// TwinCAT 3 PLC project Nepionic_Log_Test
// ProgramVersion: 3.1.4026.20
// libraries:
//   [Nepionic_Log], * (Nepionic)
//   Tc2_Standard, * (Beckhoff Automation GmbH)
//   Tc2_System, * (Beckhoff Automation GmbH)
//   Tc2_TcpIp, * (Beckhoff Automation GmbH)
//   Tc2_Utilities, * (Beckhoff Automation GmbH)
//   Tc3_Module, * (Beckhoff Automation GmbH)
// project tree:
//   Lib/ AnyToString.TcPOU, Constants.TcGVL, DateTime.TcPOU, DeleteFilesState.TcDUT, DeleteOldFiles.TcPOU, DynamicStringBuffer.TcPOU, Error.TcDUT, ErrorCodes.TcDUT, GenerateTimeData.TcPOU, GetFileAgeInSeconds.TcPOU, ILimitedStringBuilder.TcIO, ILog.TcIO, ILogCore.TcIO, IStringBuilder.TcIO, LoggingConfiguration.TcDUT, LogLevel.TcDUT, LogLevelToAdsLogMsgType.TcPOU, PersistToFileState.TcDUT, RollingIntervals.TcDUT, StringBuilder.TcPOU, TcLog.TcPOU, TcLogCore.TcPOU, TcLogTrig.TcPOU
//   Lib/Syslog/ SyslogClient.TcPOU
//   Programs/ TestRunner.TcPOU
//   Tasks/ TestTask.TcTTO
// real-time tasks:
//   TASK PlcTask: cycle T#10ms, priority 20, ADS port 350

CONFIGURATION Nepionic_Log_Test
    RESOURCE PLC ON TwinCAT3
        TASK TestTask(INTERVAL := T#10ms, PRIORITY := 20);
        PROGRAM TestRunner WITH TestTask : TestRunner;
    END_RESOURCE
END_CONFIGURATION

// ---- Lib/DeleteFilesState.TcDUT
// States for state machine used in `DeleteOldFiles`.
{attribute 'qualified_only'}
{attribute 'strict'}
TYPE INTERNAL DeleteFilesState :
(
	Idle := 0,
  SearchNextFile,
  WaitUntilExecutionDone,
  ProcessFoundFiles,
  CheckIfFileIsDirectory,
  CheckFileTime,
  DeleteFile,
  FileDeleted
);
END_TYPE

// ---- Lib/Error.TcDUT
/// This is the error type used in this library.
TYPE Error :
STRUCT
  /// `TRUE` signals an active error
	Active : BOOL;
  /// Error code of type `ErrorCodes`
	Code : INT;
  /// Plain text error message
	Info : Tc2_System.T_MaxString;
END_STRUCT
END_TYPE

// ---- Lib/ErrorCodes.TcDUT
/// Provides error codes for TcLogCore
{attribute 'qualified_only'}
{attribute 'strict'}
{attribute 'to_string'}
TYPE ErrorCodes : 
(
	None := 0,
	OpeningFileFailed,
	WritingToFileFailed,
	ClosingFileFailed,
	EnumeratingFilesInSpecifiedDirectoryFailed,
	DeletingFileFailed,
	FifoOverflow
);
END_TYPE

// ---- Lib/LoggingConfiguration.TcDUT
// Configuration of TcLogCore
TYPE LoggingConfiguration :
STRUCT
	// File name where the logs should be written to. Should not include path.
	file_name : Tc2_System.T_MaxString;
  // File path where the logs should be written to. Will be prefixed to `FileName`
	file_path : Tc2_System.T_MaxString;
  // Whether to include the instance path of TcLog into the log message or not.
	IncludeInstancePath : BOOL;
  /// Whether to write the logs to ADS output or not.
	WriteToAds : BOOL;
  /// Rolling interval: when to create a new log file.
	RollingInterval : RollingIntervals;
  /// What is the minimum log level that gets logged?
	MinimumLevel : LogLevel;
  /// Which delimiter should be used between the different parts of the log string?
	Delimiter : STRING(1);
  /// When should old log files be deleted? Unit: days. Set it to `0` if log files should never be deleted. 
	LogFileLifespan : UINT;
  /// Format of timestamp. See `TcLogCore.TimestampFormat` for formatting options.
	TimestampFormat : STRING;
  /// Log only valid timestamps (skip log messages during time initialization (first few cycles)
  	ValidTimestampsOnly: BOOL;
END_STRUCT
END_TYPE

// ---- Lib/LogLevel.TcDUT
{attribute 'qualified_only'}
{attribute 'strict'}
{attribute 'to_string'}
TYPE LogLevel :
(
	Debug := 0,
	Information,
	Warning,
	Error,
	Fatal
);
END_TYPE

// ---- Lib/PersistToFileState.TcDUT
// States for state machine used in `DynamicStringBuffer.PersistToFile`
{attribute 'qualified_only'}
{attribute 'strict'}
TYPE INTERNAL PersistToFileState :
(
	Idle := 0,
	OpenFile,
	GetStringFromFifo,
	AppendDataToFile,
	CloseFile
);
END_TYPE

// ---- Lib/RollingIntervals.TcDUT
/// Rolling interval to create a new log file when expired. 
{attribute 'qualified_only'}
{attribute 'strict'}
{attrivute 'to_string'}
TYPE RollingIntervals :
(
	None := 0,
	Hourly,
	Daily,
	Monthly
);
END_TYPE

// ---- Lib/Constants.TcGVL
{attribute 'qualified_only'}
VAR_GLOBAL CONSTANT
	/// Fifo overhead needed to manage the string buffer
	FifoOverhead : UDINT := 10;
	/// Buffer size of temporary buffer used to persist all log messages in one cycle. 
	BufferSize : UDINT := (100 * (Tc2_System.MAX_STRING_LENGTH + FifoOverhead));
END_VAR

// ---- Lib/ILimitedStringBuilder.TcIO
{attribute 'hide'}
INTERFACE INTERNAL ILimitedStringBuilder

METHOD Append : IStringBuilder // Append text TO t current build STRING.
VAR_INPUT
    Text : Tc2_System.T_MaxString; //Text to append to current build string
END_VAR
END_METHOD

METHOD AppendIf : IStringBuilder
VAR_INPUT
    Condition : BOOL;
    Text : Tc2_System.T_MaxString;
END_VAR
END_METHOD

METHOD Reset : ILimitedStringBuilder //Reset current build STRING TO an empty STRING.
END_METHOD

METHOD ToString : Tc2_System.T_MaxString //Returns current build STRING.
END_METHOD

END_INTERFACE

// ---- Lib/ILog.TcIO
INTERFACE ILog

METHOD SetLogger : BOOL
VAR_INPUT
    ref2Core : ILogCore;
END_VAR
END_METHOD

END_INTERFACE

// ---- Lib/ILogCore.TcIO
INTERFACE ILogCore EXTENDS __System.IQueryInterface

// Logger method.
// Logs data in custom format. No additional formatting will be done.
METHOD LogCustomFormat : BOOL
VAR_INPUT
    data : Tc2_System.T_MaxString; // Data to be logged. No additional formatting will be done.
END_VAR
END_METHOD

// Logger method.
// Logs in the standard format. This includes
// - timestamp
// - log level
// - log message
// - instance path of logging source (optional)
// The message will only be logged if the logging level exceeds the configured minimum logging level.
METHOD LogStandardFormat : BOOL
VAR_INPUT
    data : Tc2_System.T_MaxString; // Data to be logged. Additional formatting wil be done.
    instancePath : Tc2_System.T_MaxString; // Instance path of calling logger to locate source of logging message.
    logLevel : LogLevels; // Log level of message.
END_VAR
END_METHOD

END_INTERFACE

// ---- Lib/IStringBuilder.TcIO
{attribute 'hide'}
INTERFACE INTERNAL IStringBuilder

METHOD Append : IStringBuilder // Append text TO t current build STRING.
VAR_INPUT
    Text : Tc2_System.T_MaxString; //Text to append to current build string
END_VAR
END_METHOD

METHOD AppendIf : IStringBuilder
VAR_INPUT
    Condition : BOOL;
    Text : Tc2_System.T_MaxString;
END_VAR
END_METHOD

METHOD InsertAtLocation : IStringBuilder
VAR_INPUT
    Text : Tc2_System.T_MaxString;
    Position : INT;
END_VAR
END_METHOD

METHOD PadLeft : IStringBuilder
VAR_INPUT
    text : Tc2_System.T_MaxString; // Text to append to current build string
    length : INT; // Total length of text + padding
    c : STRING(1); // Character to be padded left of text
END_VAR
END_METHOD

METHOD Reset : ILimitedStringBuilder //Reset current build STRING TO an empty STRING.
END_METHOD

METHOD ToString : Tc2_System.T_MaxString //Returns current build STRING.
END_METHOD

END_INTERFACE

// ---- Programs/TestRunner.TcPOU
PROGRAM TestRunner
VAR
	syslogger : SyslogClient(hostname := '127.0.0.1', port := 514);
	
	message : STRING(255) := 'Get a hot dog up ya!';
	send : BOOL;
END_VAR

IF send THEN
	send := FALSE;
	syslogger.SendLog(2, message);
END_IF

syslogger.Execute();

END_PROGRAM

// ---- Lib/Syslog/SyslogClient.TcPOU
FUNCTION_BLOCK SyslogClient
VAR
	// Properties
	_hostname : STRING := '127.0.0.1';
	_port : UINT := 514;
	app_name : STRING(32) := 'TwinCAT_PLC';
    
	// Internal Logic
	socket_handle : Tc2_TcpIp.T_HSocket;
	socket_create : Tc2_TcpIp.Fb_SocketUdpCreate;
	udp_send : Tc2_TcpIp.Fb_SocketUdpSendTo;
    
    log_payload : STRING(512);
    timestamp : STRING(32);
    get_time : Tc2_Utilities.NT_GetTime;
    
    state : INT := 0;
END_VAR

PROPERTY PUBLIC AppName : STRING(255)
GET // PUBLIC
AppName := app_name;
END_GET
SET // PUBLIC
app_name := AppName;
END_SET
END_PROPERTY

METHOD PUBLIC Execute
CASE state OF
    0: // Idle
        
    10: // Fetch Timestamp
        get_time(START := TRUE);
        IF NOT get_time.BUSY AND NOT get_time.ERR THEN
            UpdateTimestamp();
            get_time(START := FALSE);
            state := 20;
        ELSIF get_time.ERR THEN
            get_time(START := FALSE);
            state := 0;
        END_IF

    20: // Maintain Socket
        IF socket_handle.handle = 0 THEN
			socket_create(
				bExecute := TRUE,
				sLocalHost := _hostname,
				nLocalPort := 4444
			);
			IF NOT socket_create.bBusy AND NOT socket_create.bError THEN
				socket_handle := socket_create.hSocket;
				socket_create(bExecute := FALSE);
			END_IF
		ELSE
			state := 30;
		END_IF

    30: // Dispatch UDP
        udp_send(
            hSocket := socket_handle, 
            sRemoteHost := _hostname, 
            nRemotePort := _port,
            pSrc := ADR(log_payload), 
            cbLen := INT_TO_UDINT(Tc2_Standard.Len(log_payload)), 
            bExecute := TRUE
		);
            
        IF NOT udp_send.bBusy AND NOT udp_send.bError THEN
            udp_send(bExecute := FALSE);
            state := 0; 
        END_IF
END_CASE
END_METHOD

//FB_Init is always available implicitly and it is used primarily for initialization.
//The return value is not evaluated. For a specific influence, you can also declare the
//methods explicitly and provide additional code there with the standard initialization
//code. You can evaluate the return value.
METHOD FB_Init: BOOL
VAR_INPUT
    bInitRetains: BOOL; // TRUE: the retain variables are initialized (reset warm / reset cold)
    bInCopyCode: BOOL;  // TRUE: the instance will be copied to the copy code afterward (online change)
	hostname : STRING(15);
	port : UINT;   
END_VAR
THIS^._hostname := hostname;
THIS^._port := port;
END_METHOD

PROPERTY PUBLIC Hostname : STRING(15)
GET // PUBLIC
Hostname := _hostname;
END_GET
SET // PUBLIC
_hostname := Hostname;
ResetConnection();
END_SET
END_PROPERTY

PROPERTY PUBLIC Port : UINT
GET // PUBLIC
Port := _port;
END_GET
SET // PUBLIC
_port := Port;
ResetConnection();
END_SET
END_PROPERTY

METHOD PRIVATE ResetConnection
END_METHOD

METHOD PUBLIC SendLog
VAR_INPUT
    severity : INT; // 0: Emerg ... 7: Debug
    message  : STRING(255);
END_VAR
VAR_INST
    priority : INT;
END_VAR
// Facility 1 (User) * 8 + severity
priority := 8 + severity;

// Build RFC 5424 String: <PRI>1 TIMESTAMP HOSTNAME APPNAME - - - MESSAGE
log_payload := Tc2_System.Concat('<', INT_TO_STRING(priority));
log_payload := Tc2_System.Concat(log_payload, '>1 ');
log_payload := Tc2_System.Concat(log_payload, timestamp);
log_payload := Tc2_System.Concat(log_payload, ' ');
log_payload := Tc2_System.Concat(log_payload, hostname);
log_payload := Tc2_System.Concat(log_payload, ' ');
log_payload := Tc2_System.Concat(log_payload, app_name);
log_payload := Tc2_System.Concat(log_payload, ' - - - ');
log_payload := Tc2_System.Concat(log_payload, message);

state := 10;
END_METHOD

METHOD PRIVATE UpdateTimestamp
timestamp := WORD_TO_STRING(get_time.TimeStr.wYear);
timestamp := Tc2_System.Concat(timestamp, '-');
timestamp := Tc2_System.Concat(timestamp, Tc2_System.RIGHT(Tc2_System.Concat('0', WORD_TO_STRING(get_time.TimeStr.wMonth)), 2));
timestamp := Tc2_System.Concat(timestamp, '-');
timestamp := Tc2_System.Concat(timestamp, Tc2_System.RIGHT(Tc2_System.Concat('0', WORD_TO_STRING(get_time.TimeStr.wDay)), 2));
timestamp := Tc2_System.Concat(timestamp, 'T');
timestamp := Tc2_System.Concat(timestamp, Tc2_System.RIGHT(Tc2_System.Concat('0', WORD_TO_STRING(get_time.TimeStr.wHour)), 2));
timestamp := Tc2_System.Concat(timestamp, ':');
timestamp := Tc2_System.Concat(timestamp, Tc2_System.RIGHT(Tc2_System.Concat('0', WORD_TO_STRING(get_time.TimeStr.wMinute)), 2));
timestamp := Tc2_System.Concat(timestamp, ':');
timestamp := Tc2_System.Concat(timestamp, Tc2_System.RIGHT(Tc2_System.Concat('0', WORD_TO_STRING(get_time.TimeStr.wSecond)), 2));
timestamp := Tc2_System.Concat(timestamp, 'Z');
END_METHOD

END_FUNCTION_BLOCK

// ---- Lib/AnyToString.TcPOU
/// Converts value of input data to string, where the input type can be any of 
/// the standard data types.
FUNCTION PUBLIC AnyToString : Tc2_System.T_MaxString
VAR_INPUT
	data : ANY;
END_VAR
VAR
	_any_byte : POINTER TO BYTE;
	_any_usint : POINTER TO USINT;
	_any_int : POINTER TO INT;
	_any_uint : POINTER TO UINT;
	_any_udInt : POINTER TO UDINT;
	_any_sint : POINTER TO SINT;
	_any_dint : POINTER TO DINT;
	_any_lint : POINTER TO LINT;
	_any_ulint : POINTER TO ULINT;
	_any_word : POINTER TO WORD;
	_any_lword : POINTER TO LWORD;
	_any_real : POINTER TO REAL;
	_any_lreal : POINTER TO LREAL;
	_any_date_and_time : POINTER TO DATE_AND_TIME;
	_any_date : POINTER TO DATE;
	_any_time : POINTER TO TIME;
	_any_wstring : POINTER TO WSTRING;
	_any_time_of_day : POINTER TO TOD;
	_any_string : POINTER TO STRING;
	_string : Tc2_System.T_MaxString;
	_wstring : WSTRING;
END_VAR

IF data.TypeClass = __SYSTEM.Type_Class.Type_Byte THEN
	_any_byte := data.pValue;
	AnyToString := BYTE_TO_STRING(_any_byte^);
ELSIF data.TypeClass = __SYSTEM.Type_Class.Type_Int THEN
	_any_int := data.pValue;
	AnyToString := INT_TO_STRING(_any_int^);
ELSIF data.TypeClass = __SYSTEM.Type_Class.Type_UInt THEN
	_any_uint := data.pValue;
	AnyToString := UINT_TO_STRING(_any_uint^);
ELSIF data.TypeClass = __SYSTEM.Type_Class.Type_UDint THEN
	_any_udint := data.pValue;
	AnyToString := UDINT_TO_STRING(_any_udint^);
ELSIF data.TypeClass = __SYSTEM.Type_Class.Type_SInt THEN
	_any_sint := data.pValue;
	AnyToString := SINT_TO_STRING(_any_sint^);
ELSIF data.TypeClass = __SYSTEM.Type_Class.Type_USint THEN
	_any_usint := data.pValue;
	AnyToString := USINT_TO_STRING(_any_usint^);
ELSIF data.TypeClass = __SYSTEM.Type_Class.Type_DInt THEN
	_any_dint := data.pValue;
	AnyToString := DINT_TO_STRING(_any_dint^);
ELSIF data.TypeClass = __SYSTEM.Type_Class.Type_LInt THEN
	_any_lint := data.pValue;
	AnyToString := LINT_TO_STRING(_any_lint^);
ELSIF data.TypeClass = __SYSTEM.Type_Class.Type_ULint THEN
	_any_ulint := data.pValue;
	AnyToString := ULINT_TO_STRING(_any_ulint^);
ELSIF data.TypeClass = __SYSTEM.Type_Class.Type_Word THEN
	_any_word := data.pValue;
	AnyToString := WORD_TO_STRING(_any_word^);
ELSIF data.TypeClass = __SYSTEM.Type_Class.Type_LWord THEN
	_any_lword := data.pValue;
	AnyToString := LWORD_TO_STRING(_any_lword^);
ELSIF data.TypeClass = __SYSTEM.Type_Class.Type_Real THEN
	_any_real := data.pValue;
	AnyToString := REAL_TO_STRING(_any_real^);
ELSIF data.TypeClass = __SYSTEM.Type_Class.Type_LReal THEN
	_any_lreal := data.pValue;
	AnyToString := LREAL_TO_STRING(_any_lreal^);
ELSIF data.TypeClass = __SYSTEM.Type_Class.Type_DateAndTime THEN
	_any_date_and_time := data.pValue;
	AnyToString := DT_TO_STRING(_any_date_and_time^);  
ELSIF data.TypeClass = __SYSTEM.Type_Class.Type_Date THEN
	_any_date := data.pValue;
	AnyToString := DATE_TO_STRING(_any_date^);
ELSIF data.TypeClass = __SYSTEM.Type_Class.Type_Time THEN
	_any_time := data.pValue;
	AnyToString := TIME_TO_STRING(_any_time^);
ELSIF data.TypeClass = __SYSTEM.Type_Class.Type_String THEN
	_any_string := data.pValue;
	AnyToString := _any_string^;
ELSIF data.TypeClass = __SYSTEM.Type_Class.Type_WString THEN
	_any_wstring := data.pValue;
	_wString := _any_wstring^;
	Tc2_Utilities.WSTRING_TO_STRING2(ADR(_string), ADR(_wstring), SIZEOF(_wstring));
	AnyToString := _string;
ELSIF data.TypeClass = __SYSTEM.Type_Class.Type_TimeOfDay THEN
	_any_time_of_day := data.pValue;
	AnyToString := TOD_TO_STRING(_any_time_of_day^);
ELSE
	AnyToString := TO_STRING(data.pValue^);
END_IF

END_FUNCTION

// ---- Lib/DateTime.TcPOU
/// Generate time data in different formats.
{attribute: 'hide_all_locals'}
FUNCTION_BLOCK PUBLIC DateTime
VAR
  local_system_time : Tc2_Utilities.FB_LocalSystemTime;
  get_system_time : Tc2_System.GetSystemTime;
  time_zone_info : Tc2_Utilities.FB_GetTimeZoneInformation;
  local_Time : Tc2_Utilities.FB_SystemTimeToTzSpecificLocalTime;
  local_system_time_valid : Tc2_Standard.R_Trig;
  utc_time : Tc2_Utilities.FB_TzSpecificLocalTimeToFileTime;
END_VAR

// Get local system time
local_system_time(
	sNetID  :=  '',
	bEnable :=  TRUE,
	dwCycle :=  1,
	dwOpt :=  1,
	tTimeout:= Tc2_System.Default_Ads_Timeout
);

// Get timezone information
time_zone_info(
	sNetID := '',
	bExecute := TRUE,
	tTimeout := Tc2_System.Default_Ads_Timeout
);

// Convert local time to utc time
utc_time(
	in := THIS^.AsLocalFileTime,
	tzInfo := time_zone_info.tzInfo
);
  
// Finished retrieving time data
local_system_time_valid(Clk := local_system_time.bValid);

/// Returns local time as `Tc2_Utilities.T_FILETIME`.
{attribute 'monitoring':='variable'}
PROPERTY AsLocalFileTime : Tc2_Utilities.T_FILETIME
GET
AsLocalFileTime := SYSTEMTIME_TO_FILETIME(THIS^.AsLocalSystemTime);
END_GET
END_PROPERTY

/// Returns local time as `Tc2_Utilities.TIMESTRUCT`.
{attribute 'monitoring':='variable'}
PROPERTY AsLocalSystemTime : Tc2_Utilities.TIMESTRUCT
GET
AsLocalSystemTime := local_system_time.systemTime;
END_GET
END_PROPERTY

/// Returns local time as string.
{attribute 'monitoring':='variable'}
PROPERTY AsLocalSystemTimeString : Tc2_System.T_MAXSTRING
GET
AsLocalSystemTimeString := Tc2_Utilities.SYSTEMTIME_TO_STRING(THIS^.AsLocalSystemTime);
END_GET
END_PROPERTY

/// Returns UTC time as `Tc2_Utilities.T_FILETIME`.
{attribute 'monitoring':='variable'}
PROPERTY AsUtcFileTime : Tc2_Utilities.T_FILETIME
GET
AsUtcFileTime := utc_time.out;
END_GET
END_PROPERTY

/// When calling `DateTime` the first time, it takes some time until all time and timezone information is available.
/// `Done` is `TRUE` for one cycle, once all the data is ready. 
{attribute 'monitoring':='call'}
PROPERTY Done : BOOL
GET
Done := local_system_time_valid.Q;
END_GET
END_PROPERTY

// Replaces placeholders in format string by the actual time values.
{attribute 'hide_all_locals'}
{attribute 'hide'}
METHOD PRIVATE ReplaceFormatPlaceholder : STRING
VAR_INPUT
  format : STRING;
  length : INT;
  timeType : STRING(1);
END_VAR
VAR_INST
  i : INT;
  replaceString : STRING;
  timeString : STRING;
END_VAR
VAR
  localSystemTime : Tc2_Utilities.TIMESTRUCT;
END_VAR
localSystemTime := THIS^.AsLocalSystemTime;

IF    timeType = 'Y'  THEN timeString := TO_STRING(localSystemTime.wYear); 
ELSIF timeType = 'M'  THEN timeString := TO_STRING(localSystemTime.wMonth); 
ELSIF timeType = 'D'  THEN timeString := TO_STRING(localSystemTime.wDay); 
ELSIF timeType = 'h'  THEN timeString := TO_STRING(localSystemTime.wHour); 
ELSIF timeType = 'm'  THEN timeString := TO_STRING(localSystemTime.wMinute); 
ELSIF timeType = 's'  THEN timeString := TO_STRING(localSystemTime.wSecond); 
ELSIF timeType = 'i'  THEN timeString := TO_STRING(localSystemTime.wMilliseconds); 
ELSE
  timeString:='';
END_IF

replaceString := '';

IF length > Tc2_Standard.LEN(timeString) THEN
  FOR i:=1 TO length - Tc2_Standard.LEN(timeString) DO
    replaceString := Tc2_Standard.CONCAT(replaceString, '0');
  END_FOR
  replaceString := Tc2_Standard.CONCAT(replaceString, timeString);
ELSE
  replaceString := Tc2_Standard.RIGHT(timeString, length);
END_IF

ReplaceFormatPlaceholder := Tc2_Standard.REPLACE(format, replaceString, length, Tc2_Standard.FIND(format, timeType));
END_METHOD

/// Returns a formatted string containing the actual time information 
/// - `Y` : year
/// - `M` : month
/// - `D` : day
/// - `h` : hour 
/// - `m` : minute
/// - `s` : second
/// - `i` : millisecond
/// 
/// Example:    
/// _YYMMDD-hh:mm:ss:iii_   
/// => _20210812-12:30:22:123_
{attribute 'hide_all_locals'}
METHOD ToFormatString : Tc2_System.T_MaxString
VAR_INPUT
  /// Format the timestamp should have.
  format : STRING;
END_VAR
VAR_INST
  inputString : STRING;
  c : STRING(1);
  formattedString : Tc2_System.T_MaxString;
END_VAR
VAR
  year : INT := 0;
  month : INT := 0;
  day : INT := 0;
  hour : INT := 0;
  minute : INT := 0;
  second : INT := 0;
  millisecond : INT := 0;
END_VAR
VAR CONSTANT
  ValidFormat : STRING := 'YMDhms';
END_VAR
// Parses "format" and returns a adequatly formatted string containing the time information
inputString := format;

WHILE Tc2_Standard.LEN(inputString) > 0 DO
  c := Tc2_Standard.LEFT(inputString, 1);
  
  IF    c = 'Y' THEN year := year + 1;
  ELSIF c = 'M' THEN month := month + 1;
  ELSIF c = 'D' THEN day := day + 1;
  ELSIF c = 'h' THEN hour := hour + 1;
  ELSIF c = 'm' THEN minute := minute + 1;
  ELSIF c = 's' THEN second := second + 1;
  ELSIF c = 'i' THEN millisecond := millisecond + 1;
  END_IF
  
  inputString := Tc2_Standard.DELETE(inputString, 1, 1);
END_WHILE

formattedString := ReplaceFormatPlaceholder(format, year, 'Y');
formattedString := ReplaceFormatPlaceholder(formattedString, month, 'M');
formattedString := ReplaceFormatPlaceholder(formattedString, day, 'D');
formattedString := ReplaceFormatPlaceholder(formattedString, hour, 'h');
formattedString := ReplaceFormatPlaceholder(formattedString, minute, 'm');
formattedString := ReplaceFormatPlaceholder(formattedString, second, 's');
formattedString := ReplaceFormatPlaceholder(formattedString, millisecond, 'i');

ToFormatString := formattedString;
END_METHOD

END_FUNCTION_BLOCK

// ---- Lib/DeleteOldFiles.TcPOU
{attribute 'hide_all_locals'}
FUNCTION_BLOCK INTERNAL DeleteOldFiles
VAR_INPUT
  StartScan : BOOL; // Rising edge starts scan for out-of-date log files and deletes them.
  ExpirationInDays : UINT; // Files will be deleted if older than n days
  FilePath : Tc2_System.T_MaxString; // Path to files to be deleted
  FileName : Tc2_System.T_MaxString; // Only files which match this filename will be deleted
  CurrentUtcTime : Tc2_Utilities.T_FILETIME; // Current time  as UTC
END_VAR
VAR_OUTPUT
  Error : Error; // Error information
END_VAR
VAR CONSTANT
  OneDayInSeconds : LREAL := 24*3600.0;
  MaxNumberOfFiles : UDINT := 100;
END_VAR
VAR
  _state : DeleteFilesState := DeleteFilesState.Idle;
  
  _enumFindFileList : Tc2_Utilities.FB_EnumFindFileList;
  _enumBusy : Tc2_Standard.F_TRIG;
  _fileDelete : Tc2_System.FB_FileDelete;
  _fileDeleteBusy : Tc2_Standard.F_TRIG;
  _listOfFiles : ARRAY[1..100] OF Tc2_Utilities.ST_FindFileEntry;
  _deleteFileIndex : UDINT;
  _fileNameToDelete : Tc2_System.T_MaxString;
  _commandType : Tc2_Utilities.E_EnumCmdType;
  _fileDeleted : BOOL;
  _startFileDelete: BOOL;
END_VAR

// State machine to delete all due files.
// It first enumerates all files in the specified directory
// and then deletes all files that have overpassed the specified due date
_startFileDelete := FALSE;

CASE _state OF
  DeleteFilesState.Idle:
    IF StartScan THEN
      _commandType:= eEnumCmd_First;
      _deleteFileIndex := 1;
      _state := DeleteFilesState.SearchNextFile;
    END_IF
    
  DeleteFilesState.SearchNextFile:
    IF _enumBusy.Q THEN
      _state := DeleteFilesState.WaitUntilExecutionDone;
    END_IF
    
  DeleteFilesState.WaitUntilExecutionDone:
    IF NOT _enumFindFileList.bError THEN
      IF NOT _enumFindFileList.bEOE THEN
        IF _enumFindFileList.nFindFiles < MaxNumberOfFiles THEN
          _state := DeleteFilesState.SearchNextFile;
        ELSE
          _commandType := eEnumCmd_Abort;
          _state := DeleteFilesState.ProcessFoundFiles;
        END_IF
      ELSE
        _state := DeleteFilesState.ProcessFoundFiles;
      END_IF
    ELSE
      _state := DeleteFilesState.Idle;
    END_IF
    
  DeleteFilesState.ProcessFoundFiles:
    IF _deleteFileIndex > _enumFindFileList.nFindFiles THEN
      _state := DeleteFilesState.Idle;
    ELSE
      _state := DeleteFilesState.CheckIfFileIsDirectory;
    END_IF
    
  DeleteFilesState.CheckIfFileIsDirectory:
    IF NOT _listOfFiles[_deleteFileIndex].fileAttributes.bDirectory THEN
      _state := DeleteFilesState.CheckFileTime;
    ELSE
      _deleteFileIndex := _deleteFileIndex + 1;
      _state := DeleteFilesState.ProcessFoundFiles;
    END_IF
    
  DeleteFilesState.CheckFileTime:   
    IF GetFileAgeInSeconds(CurrentUtcTime, _listOfFiles[_deleteFileIndex]) > (ExpirationInDays * OneDayInSeconds) THEN
      _state := DeleteFilesState.DeleteFile;
    ELSE
      _deleteFileIndex := _deleteFileIndex + 1;
      _state := DeleteFilesState.ProcessFoundFiles;
    END_IF
  
  DeleteFilesState.DeleteFile:
    _fileNameToDelete := Tc2_Standard.CONCAT(FilePath, _listOfFiles[_deleteFileIndex].sFileName);
    _startFileDelete := TRUE;
    
    IF _fileDeleteBusy.Q THEN
      _deleteFileIndex := _deleteFileIndex + 1;
      _fileDeleted := TRUE;
      _state := DeleteFilesState.FileDeleted;
    END_IF
    IF _fileDelete.bError THEN
      _state := DeleteFilesState.Idle;
    END_IF
    
  DeleteFilesState.FileDeleted:   
    // This state is needed to generate a rising edge for FB_FileDelete
    IF NOT _fileDeleted THEN
      _state := DeleteFilesState.ProcessFoundFiles;
    END_IF
    _fileDeleted := FALSE;

END_CASE

// Function blocks used in state machine

// Search files in given directory
_enumFindFileList(sNetId := '',
       eCmd := _commandType,
       sPathName := Tc2_Standard.CONCAT(FilePath, Tc2_Standard.CONCAT('*', FileName)),
       bExecute := (_state = DeleteFilesState.SearchNextFile) OR (_commandType = eEnumCmd_Abort AND _state <> DeleteFilesState.Idle),
       pFindList := ADR(_listOfFiles),
       cbFindList := SIZEOF(_listOfFiles),
       tTimeout := T#10S);
       
_enumBusy(CLK:=_enumFindFileList.bBusy);

// Delete files
_fileDelete(sNetId := '',
             sPathName := _fileNameToDelete,
             bExecute := _startFileDelete,
             tTimeout := T#10S);

_fileDeleteBusy(CLK := _fileDelete.bBusy);

// Error handling
Error.Active := FALSE;
Error.Code := ErrorCodes.None;
Error.Info := '';

IF _enumFindFileList.bError THEN
  Error.Active := TRUE;
  Error.Code := ErrorCodes.EnumeratingFilesInSpecifiedDirectoryFailed;
  Error.Info := Tc2_Standard.CONCAT('Enumerating files in specified directory failed. Error thrown by FB_EnumFindFileList. Consult Beckhoff InfoSys. Internal Error: ', UDINT_TO_STRING(_enumFindFileList.nErrId));
END_IF
      
IF _fileDelete.bError THEN
  Error.Active := TRUE;
  Error.Code := ErrorCodes.DeletingFileFailed;
  Error.Info := Tc2_Standard.CONCAT('Deleting expired log file in specified directory failed. Error thrown by FB_FileDelete. Consult Beckhoff InfoSys. Internal Error: ', UDINT_TO_STRING(_fileDelete.nErrId));
END_IF

END_FUNCTION_BLOCK

// ---- Lib/GetFileAgeInSeconds.TcPOU
{attribute 'hide'}
FUNCTION INTERNAL GetFileAgeInSeconds : DINT
VAR_INPUT
  currentUtcTime : Tc2_Utilities.T_FILETIME;
  findFileEntry : Tc2_Utilities.ST_FindFileEntry;
END_VAR
VAR
  _timeLastWriteAccess : Tc2_Utilities.T_ULARGE_INTEGER;
  _fileTimeAsULINT : Tc2_Utilities.T_ULARGE_INTEGER;
  _fileTimeDifference : Tc2_Utilities.T_ULARGE_INTEGER;
END_VAR
VAR CONSTANT
  OneSecondInOneHundredNanoSecondsIntervals : LREAL := 1000*1000*10;
END_VAR

// Local file time
_fileTimeAsULINT.dwLowPart := currentUtcTime.dwLowDateTime;
_fileTimeAsULINT.dwHighPart := currentUtcTime.dwHighDateTime;

// Write access is UTC
_timeLastWriteAccess.dwLowPart := findFileEntry.lastWriteTime.dwLowDateTime;
_timeLastWriteAccess.dwHighPart := findFileEntry.lastWriteTime.dwHighDateTime;
_fileTimeDifference := UInt64Sub64(_fileTimeAsULINT, _timeLastWriteAccess);

GetFileAgeInSeconds := LREAL_TO_DINT(UINT64_TO_LREAL(_fileTimeDifference)/(OneSecondInOneHundredNanoSecondsIntervals));

END_FUNCTION

// ---- Lib/DynamicStringBuffer.TcPOU
{attribute 'hide_all_locals'}
FUNCTION_BLOCK INTERNAL DynamicStringBuffer
VAR_OUTPUT
  Error : Error; // Error information of this FB
END_VAR
VAR
  _fifo : Tc2_Utilities.FB_StringRingBuffer; // Necessary to buffer log data until it has been written to file.
  _memoryManager : Tc3_DynamicMemory.FB_DynMem_Manager; // Memory manager, required by DynMem_Buffer.
  _dynamicMemoryBuffer : Tc3_DynamicMemory.FB_DynMem_Buffer(ipMemMan := _memoryManager); // Provides dynamic buffer for Fifo. Is extended automatically if more than the
                                                                   // default buffer size is needed.                  
  _busy : BOOL; // Buffer is busy; typically with writing data to the file system.
END_VAR

METHOD AddLine : BOOL
VAR_INPUT
  text : Tc2_System.T_MaxString; // Text to be added to the buffer
END_VAR
ResizeFifoBufferIfNecessary();
_fifo.A_AddTail(putValue := Tc2_Standard.CONCAT(Tc2_Standard.LEFT(text, 254), '$N'));
END_METHOD

METHOD AddString : BOOL
VAR_INPUT
  text : Tc2_System.T_MaxString; // String to be added to the buffer
END_VAR
ResizeFifoBufferIfNecessary();
_fifo.A_AddTail(putValue := text);
END_METHOD

METHOD PRIVATE AllocateBuffer : BOOL // Allocates buffer FOR the fifo.
VAR_INPUT
  bufferSize : UDINT; // Initial buffer size in BYTEs for fifo buffer.
END_VAR
_dynamicMemoryBuffer.CreateBuffer(nSize:=bufferSize, bReset:=TRUE);
_fifo.pBuffer := _dynamicMemoryBuffer.pBuffer;
_fifo.cbBuffer := bufferSize;
END_METHOD

{attribute 'monitoring':='call'}
PROPERTY Busy : BOOL
GET
Busy := _busy;
END_GET
SET // PRIVATE
_busy := Busy;
END_SET
END_PROPERTY

METHOD FB_exit : BOOL
VAR_INPUT
  bInCopyCode : BOOL; // if TRUE, the exit method is called for exiting an instance that is copied afterwards (online change).
END_VAR
_dynamicMemoryBuffer.Clear();
END_METHOD

METHOD FlushCache : BOOL
_fifo.A_Reset();
END_METHOD

METHOD INTERNAL Init : BOOL
VAR_INPUT
  bufferSize : UDINT; // Initial buffer size in BYTEs for fifo buffer.
END_VAR
AllocateBuffer(bufferSize);
END_METHOD

{attribute 'hide_all_locals'}
METHOD PersistToFile : BOOL
VAR_INPUT
  enable: BOOL; // TRUE starts persistence mechanism
  fileName : Tc2_System.T_MaxString; // File name including its path
END_VAR
VAR_INST
  state : PersistToFileState;
  
  fileOpen : Tc2_System.FB_FileOpen;
  fileHandle : UINT;
  
  fileWrite : Tc2_System.FB_FileWrite;
  lockFileWriteToForceRisingEdge : BOOL; // filePuts can only be executed every other cycle
                                         // since it needs a rising edge to execute.
  fileClose : Tc2_System.FB_FileClose;
  
  buffer : ARRAY[0..CONSTANTS.BufferSize] OF BYTE;
  currentBufferPos : UDINT;
  fifoHeadString : Tc2_System.T_MaxString;
  fifoHeadLength : UDINT;
  fifoHeadBytes : ARRAY[0..Tc2_System.MAX_STRING_LENGTH] OF BYTE;
  i : UINT;
END_VAR
VAR CONSTANT
  NetId : STRING := '';
  Timeout : TIME := DEFAULT_ADS_TIMEOUT;
  MaxLogsPerCycle : UINT := UDINT_TO_UINT(CONSTANTS.BufferSize / Tc2_System.MAX_STRING_LENGTH);
  MaxBufferPosition : UDINT := (SIZEOF(buffer)-Tc2_System.MAX_STRING_LENGTH);
END_VAR
// State machine
// Using if-statements instead of case for performance reasons:
// Some states execute instantly and allow thus the next state 
// to start within the same plc cycle.

// *** I D L E ***
IF state = PersistToFileState.Idle THEN
  lockFileWriteToForceRisingEdge := FALSE;
  IF _fifo.nCount > 0 AND enable THEN 
    lockFileWriteToForceRisingEdge := FALSE;
    state := PersistToFileState.OpenFile;
  END_IF
END_IF
    
// *** O P E N   F I L E ***
fileOpen(sNetId := NetId, sPathName := fileName, nMode := FOPEN_MODEAPPEND OR FOPEN_MODETEXT, 
           ePath := PATH_GENERIC, bExecute := (state = PersistToFileState.OpenFile), tTimeout := Timeout,
           hFile => fileHandle);

IF state = PersistToFileState.OpenFile THEN
  IF fileOpen.bError THEN
    state := PersistToFileState.CloseFile;
  ELSIF NOT fileOpen.bBusy THEN
    state := PersistToFileState.GetStringFromFifo; 
  END_IF
END_IF 

// *** P O P   F R O M   F I F O ***
IF state = PersistToFileState.GetStringFromFifo THEN
  IF NOT lockFileWriteToForceRisingEdge THEN
    currentBufferPos := 0;
    FOR i:=0 TO MaxLogsPerCycle DO
      IF _fifo.nCount <= 0 THEN EXIT; END_IF
      IF currentBufferPos >= MaxBufferPosition THEN EXIT; END_IF
      
      _fifo.A_RemoveHead(getValue => fifoHeadString); 
      fifoHeadBytes := MAXSTRING_TO_BYTEARR(fifoHeadString);
      fifoHeadLength := INT_TO_UDINT(LEN(fifoHeadString));
      MEMCPY(
        destAddr  :=  ADR(buffer) + SIZEOF(BYTE) * currentBufferPos,
        srcAddr   :=  ADR(fifoHeadBytes),
        n     :=  fifoHeadLength);    
      currentBufferPos := currentBufferPos + fifoHeadLength;  
    END_FOR
    state := PersistToFileState.AppendDataToFile;
  END_IF
  lockFileWriteToForceRisingEdge := FALSE;
END_IF
  
// *** W R I T E   T O   F I L E ***
fileWrite(
  sNetId := NetId, 
  hFile := fileHandle, 
  pWriteBuff := ADR(buffer),
  cbWriteLen := currentBufferPos,
  bExecute := state = PersistToFileState.AppendDataToFile, 
  tTimeout := Timeout); 

IF state = PersistToFileState.AppendDataToFile THEN
  lockFileWriteToForceRisingEdge := TRUE;   
  IF fileWrite.bError THEN
    state := PersistToFileState.CloseFile;
  ELSIF _fifo.nCount > 0 AND NOT fileWrite.bBusy THEN
    state := PersistToFileState.GetStringFromFifo; 
  ELSIF _fifo.nCount = 0 THEN
    state := PersistToFileState.CloseFile;
  END_IF
END_IF
    
// *** C L O S E   F I L E ***
fileClose(
  sNetId := NetId, hFile := fileHandle, 
  bExecute := (state = PersistToFileState.CloseFile), tTimeout := Timeout);

IF state = PersistToFileState.CloseFile THEN
  IF NOT fileClose.bBusy THEN state := PersistToFileState.Idle; END_IF
END_IF

// Close file in case of error
IF fileOpen.bError THEN state := PersistToFileState.CloseFile; END_IF
IF fileWrite.bError THEN state := PersistToFileState.CloseFile; END_IF
IF NOT _fifo.bOk AND _fifo.nCount > 0 AND state <> PersistToFileState.Idle THEN 
  state := PersistToFileState.CloseFile; 
END_IF

// Error handling
IF fileOpen.bError THEN
  Error.Active := TRUE;
  Error.Code := ErrorCodes.OpeningFileFailed;
  Error.Info := Tc2_Standard.CONCAT('Opening file failed. Error thrown by FB_FileOpen. Consult Beckhoff InfoSys. Internal Error: ', UDINT_TO_STRING(fileOpen.nErrId));
ELSIF fileWrite.bError THEN
  Error.Active := TRUE;
  Error.Code := ErrorCodes.WritingToFileFailed;
  Error.Info := Tc2_Standard.CONCAT('Writing to file failed. Error thrown by FB_FileWrite. Consult Beckhoff InfoSys. Internal Error: ', UDINT_TO_STRING(fileWrite.nErrId));
ELSIF fileClose.bError THEN
  Error.Active := TRUE;
  Error.Code := ErrorCodes.ClosingFileFailed;
  Error.Info := Tc2_Standard.CONCAT('Closing file failed. Error thrown by FB_FileClose. Consult Beckhoff InfoSys. Internal Error: ', UDINT_TO_STRING(fileClose.nErrId));
ELSIF NOT _fifo.bOk AND _fifo.nCount > 0 THEN
  Error.Active := TRUE;
  Error.Code := ErrorCodes.FifoOverflow;
  Error.Info := 'FIFO overflow. Check if plc has enough free memory.';
ELSE
  Error.Active := FALSE;
  Error.Code := ErrorCodes.None;
  Error.Info := '';
END_IF

// Set busy state
Busy := (state <> PersistToFileState.Idle OR _fifo.nCount > 0);

(* Uncomment for cyclic logging of state machine, buffer usage & errors

ADSLOGSTR(ADSLOG_MSGTYPE_LOG, 
  Tc2_Standard.CONCAT('****DynamicStringBuffer.state:', 
  Tc2_Standard.CONCAT(UINT_TO_STRING(state),
  Tc2_Standard.CONCAT(', DynamicStringBuffer.hFile:', UINT_TO_STRING(hFile)))), '');

ADSLOGSTR(ADSLOG_MSGTYPE_LOG, 
  Tc2_Standard.CONCAT('****Fifo: used ', 
  Tc2_Standard.CONCAT(UDINT_TO_STRING(Fifo.cbSize),
  Tc2_Standard.CONCAT(' of ', UDINT_TO_STRING(Fifo.cbBuffer)))), '');
  
IF Error.Active THEN
  ADSLOGSTR(ADSLOG_MSGTYPE_LOG, 
    Tc2_Standard.CONCAT('****DynamicStringBuffer.Error: ', Error.Info), 
    '');  
END_IF
*)
END_METHOD

METHOD PopHead : Tc2_System.T_MaxString
VAR_INST
  headString : Tc2_System.T_MaxString;
END_VAR
_fifo.A_RemoveHead(getValue => headString);
PopHead := headString;
END_METHOD

// Resizes the buffer for the FIFO if necessary
METHOD PRIVATE ResizeFifoBufferIfNecessary : BOOL
VAR
  requiredSize : UDINT;
  newSize : DINT;
END_VAR
requiredSize := _fifo.cbSize + (Tc2_System.MAX_STRING_LENGTH + Constants.FifoOverhead);

IF requiredSize > _fifo.cbBuffer THEN
  _dynamicMemoryBuffer.Resize(nSize := requiredSize*SIZEOF(BYTE), bPreserve:=TRUE, bReset:=TRUE);
  _fifo.pBuffer := _dynamicMemoryBuffer.pBuffer;
  _fifo.cbBuffer := requiredSize;
END_IF
END_METHOD

END_FUNCTION_BLOCK

// ---- Lib/GenerateTimeData.TcPOU
FUNCTION_BLOCK GenerateTimeData
VAR_OUTPUT
	timeAsFileTime : Tc2_Utilities.T_FILETIME;
	timeAsSystemTime : Tc2_Utilities.TIMESTRUCT;
	timeAsString : Tc2_System.T_MaxString;
	utcTimeAsFileTime : Tc2_Utilities.T_FILETIME;
END_VAR
VAR
	_localSystemTime : Tc2_Utilities.FB_LocalSystemTime;
	_getSystemTime : Tc2_System.GETSYSTEMTIME;
	_timeZoneInfo : Tc2_Utilities.FB_GetTimeZoneInformation;
	_localTime : Tc2_Utilities.FB_SystemTimeToTzSpecificLocalTime;
	_localSystemTimeValid : Tc2_Standard.R_TRIG;
	_utcTime : Tc2_Utilities.FB_TzSpecificLocalTimeToFileTime;
END_VAR
VAR_TEMP
	utcSystemTime : Tc2_Utilities.TIMESTRUCT;
END_VAR

_localSystemTime(
	sNetID	:=	'',
	bEnable := 	TRUE,
	dwCycle	:=	1,
	dwOpt	:=	1,
	tTimeout:=	DEFAULT_ADS_TIMEOUT
);

_timeZoneInfo(
	sNetID := '',
	bExecute := TRUE,
	tTimeout := DEFAULT_ADS_TIMEOUT);

_UtcTime(
	in := SYSTEMTIME_TO_FILETIME(timeAsSystemTime),
	tzInfo := _timeZoneInfo.tzInfo);
	
timeAsSystemTime 	:=	_localSystemTime.systemTime;
timeAsFileTime 		:= 	SYSTEMTIME_TO_FILETIME(timeAsSystemTime);
timeAsString 		:= 	SYSTEMTIME_TO_STRING(timeAsSystemTime);
utcTimeAsFileTime	:= 	_utcTime.out;

_localSystemTimeValid(CLK := _localSystemTime.bValid);

{attribute 'monitoring':='call'}
PROPERTY Done : BOOL
GET
Done := _localSystemTimeValid.Q;
END_GET
END_PROPERTY

// Replaces placeholders in format string by the actual time values
METHOD PRIVATE ReplaceFormatPlaceholder : STRING
VAR_INPUT
	Format : STRING;
	Length : INT;
	TimeType : STRING(1);
END_VAR
VAR_INST
	i : INT;
	replaceString : STRING;
	timeString : STRING;
END_VAR
IF    TimeType = 'Y' 	THEN timeString := TO_STRING(timeAsSystemTime.wYear); 
ELSIF TimeType = 'M' 	THEN timeString := TO_STRING(timeAsSystemTime.wMonth); 
ELSIF TimeType = 'D' 	THEN timeString := TO_STRING(timeAsSystemTime.wDay); 
ELSIF TimeType = 'h' 	THEN timeString := TO_STRING(timeAsSystemTime.wHour); 
ELSIF TimeType = 'm' 	THEN timeString := TO_STRING(timeAsSystemTime.wMinute); 
ELSIF TimeType = 's' 	THEN timeString := TO_STRING(timeAsSystemTime.wSecond); 
ELSIF TimeType = 'i' 	THEN timeString := TO_STRING(timeAsSystemTime.wMilliseconds); 
ELSE
  timeString:='';
END_IF

replaceString := '';

IF Length > LEN(timeString) THEN
	FOR i:=1 TO Length - LEN(timeString) DO
		replaceString := Tc2_Standard.CONCAT(replaceString, '0');
	END_FOR
	replaceString := Tc2_Standard.CONCAT(replaceString, timeString);
ELSE
	replaceString := RIGHT(timeString, Length);
END_IF

ReplaceFormatPlaceholder := REPLACE(Format, replaceString, Length, FIND(Format, TimeType));
END_METHOD

// Returns a formatted string containing the actual time information 
//	Y : year
//	M : month
// 	D : day
//  h : hour 
//  m : minute
//  s : second
//  i : millisecond
// 
// Example: _YYMMDD-hh:mm:ss:iii_
// => _20210812-12:30:22:123_
METHOD ToString : Tc2_System.T_MaxString
VAR_INPUT
	Format : STRING;
END_VAR
VAR_INST
	inputString : STRING;
	char : STRING(1);
	formattedString : Tc2_System.T_MaxString;
END_VAR
VAR
	year : INT := 0;
	month : INT := 0;
	day : INT := 0;
	hour : INT := 0;
	minute : INT := 0;
	second : INT := 0;
	millisecond : INT := 0;
END_VAR
VAR CONSTANT
	VALID_FORMAT : STRING := 'YMDhms';
END_VAR
// Parses "Format" and returns a adequatly formatted string containing the time information
inputString := Format;

WHILE LEN(inputString) > 0 DO
	char := LEFT(inputString, 1);
	
	IF    char = 'Y' THEN 	year := year + 1;
	ELSIF char = 'M' THEN	month := month + 1;
	ELSIF char = 'D' THEN	day := day + 1;
	ELSIF char = 'h' THEN	hour := hour + 1;
	ELSIF char = 'm' THEN	minute := minute + 1;
	ELSIF char = 's' THEN 	second := second + 1;
	ELSIF char = 'i' THEN 	millisecond := millisecond + 1;
	END_IF
	
	inputString := DELETE(inputString, 1, 1);
END_WHILE

formattedString := ReplaceFormatPlaceholder(Format, year, 'Y');
formattedString := ReplaceFormatPlaceholder(formattedString, month, 'M');
formattedString := ReplaceFormatPlaceholder(formattedString, day, 'D');
formattedString := ReplaceFormatPlaceholder(formattedString, hour, 'h');
formattedString := ReplaceFormatPlaceholder(formattedString, minute, 'm');
formattedString := ReplaceFormatPlaceholder(formattedString, second, 's');
formattedString := ReplaceFormatPlaceholder(formattedString, millisecond, 'i');

ToString := formattedString;
END_METHOD

END_FUNCTION_BLOCK

// ---- Lib/LogLevelToAdsLogMsgType.TcPOU
// Converts TcLog.LogLevels into Tc2_System.AdsLog_MsgType_*.
{attribute 'hide'}
FUNCTION INTERNAL LogLevelToAdsLogMsgType : DWORD
VAR_INPUT
  log_level : LogLevel;
END_VAR
VAR
  return_value : DWORD;
END_VAR

CASE log_level OF
  LogLevel.Debug, LogLevel.Information:
    return_value := Tc2_System.AdsLog_MsgType_Hint;
  LogLevel.Warning:
    return_value := Tc2_System.AdsLog_MsgType_Warn;
  LogLevel.Error, LogLevel.Fatal:
    return_value := Tc2_System.AdsLog_MsgType_Eerror;
  ELSE
    return_value := Tc2_System.AdsLog_MsgType_Hint;
END_CASE

LogLevelToAdsLogMsgType := return_value;

END_FUNCTION

// ---- Lib/StringBuilder.TcPOU
FUNCTION_BLOCK INTERNAL StringBuilder IMPLEMENTS IStringBuilder, ILimitedStringBuilder
VAR
  {attribute 'hide'}
  _workString : Tc2_System.T_MaxString;
END_VAR

METHOD PUBLIC Append : IStringBuilder // Append text TO t current build STRING.
VAR_INPUT
  text : Tc2_System.T_MaxString; //text to append to current build string
END_VAR
_workString:= Tc2_Standard.CONCAT(_workString,text);
Append := THIS^;
END_METHOD

METHOD PUBLIC AppendIf : IStringBuilder
VAR_INPUT
  condition : BOOL;
  text : Tc2_System.T_MaxString;
END_VAR
IF condition THEN
  _workString:= Tc2_Standard.CONCAT(_workString,text);
END_IF
AppendIf := THIS^;
END_METHOD

METHOD PUBLIC InsertAtLocation : IStringBuilder
VAR_INPUT
  text : Tc2_System.T_MaxString;
  position : INT;
END_VAR
_workString := Tc2_Standard.INSERT(_workSTring,text,position);
InsertAtLocation  := THIS^;
END_METHOD

METHOD PadLeft : IStringBuilder
VAR_INPUT
  text : Tc2_System.T_MaxString; // Text to append to current build string
  length : INT; // Total length of text + padding
  c : STRING(1); // Character to be padded left of text
END_VAR
VAR
  i : INT;
  padLength : INT;
END_VAR
// Add left padding
padLength := Tc2_Standard.LEN(text) - length;
FOR i := 1 TO padLength DO
  _workString:= Tc2_Standard.CONCAT(_workString, c);
END_FOR

// Add text
_workString:= Tc2_Standard.CONCAT(_workString,text);

PadLeft := THIS^;
END_METHOD

METHOD PUBLIC Reset : ILimitedStringBuilder //Reset current build STRING TO an empty STRING.
_workString:='';
Reset := THIS^;
END_METHOD

METHOD PUBLIC ToString : Tc2_System.T_MaxString //Returns current build STRING.
ToString := _workString;
END_METHOD

END_FUNCTION_BLOCK

// ---- Lib/TcLog.TcPOU
/// `TcLog` is the client side of the logger.  
///
/// It is used to send the logs to `TcLogCore`. Typically, it is instantiated
/// once in each `FUNCTION_BLOCK` or `PROGRAM` where logging is done. The same 
/// instance can then be used for all logging within that POU. 
///
/// `TcLog` implements a string builder that facilitates the compilation of the log
/// message without the need for external data type conversions or multiple chained `CONCAT` calls.
/// See the method section for more information.
///
/// The last method to call after the log message has been built is one of ´[Debug|Information|Warning|Error|Fatal]`. 
/// This sets the log level of the message and sends it off to the log message queue of `TcLogCore` where it will
/// be processed according to its configuration.
{attribute 'hide_all_locals'}
{attribute 'reflection'} 
FUNCTION_BLOCK TcLog IMPLEMENTS ILog
VAR
  _logConditionSatisfied : BOOL; // flag that indicates, whether log condition has been satisfied.
                                // Logging will only be carried out it this evaluates to TRUE.                    
  _logDataInitialized : BOOL; // flag that indicate, whether log data has been initialized.
                             // Necessary for configuration methods to provide a fluent interface.                            
  _logData : Tc2_System.T_MaxString; // contains message to be logged.
  _usedLogger : ILogCore;
  {attribute 'instance-path'} 
  {attribute 'noinit'} 
  _instancePath : STRING; // contains instance path
END_VAR
VAR_STAT
  {attribute 'hide'}
  s_loggerSingletonInstance : ILogCore; // Wires up TcLog ("Client") to TcLogCore ("Server") (Singleton-Behaviour)
END_VAR
VAR CONSTANT
  InvalidLoggerReference : UDINT := 0;
END_VAR

/// Appends any given data to the log string. The type of the provided data
/// has to be one of the [standard data types](https://infosys.beckhoff.com/english.php?content=../content/1033/tc3_plc_intro/2529388939.html&id=).
/// This method can be chained.
METHOD AppendAny : REFERENCE TO TcLog
VAR_INPUT
  /// data to be appended to log string.
  data : ANY;
END_VAR
InitializeLogData();

_logData := Tc2_Standard.CONCAT(_logData, AnyToString(data));

AppendAny REF= THIS^;
END_METHOD

/// Appends another string to the log message.
/// This method can be chained.
METHOD AppendString : REFERENCE TO TcLog
VAR_INPUT
  /// data to be appended to log string.
  data : Tc2_System.T_MaxString; 
END_VAR
InitializeLogData();

_logData := Tc2_Standard.CONCAT(_logData, data);
  
AppendString REF= THIS^;
END_METHOD

/// Appends information about the given variable to the log string. 
/// This method can be chained.
/// Example: 

/// ```st
/// VAR
///   Logger: TcLog;
///    myInt : INT := 10;
///   myVarInfo : __SYSTEM.VAR_INFO := __VARINFO(myInt);
/// END_VAR
/// Logger.AppendVariable(myVarInfo, myInt);
/// ```
///
METHOD AppendVariable : REFERENCE TO TcLog
VAR_INPUT
  /// [VAR_INFO](https://infosys.beckhoff.com/index.php?content=../content/1031/tc3_plc_intro/3527777675.html&id=) of variable to be appended to log string.
  varInfo : __SYSTEM.VAR_INFO;
  /// Value of variable to be appended to log string.
  value : ANY; 
END_VAR
VAR
  format : Tc2_Utilities.FB_FormatString;
  symbolName : Tc2_System.T_MaxString;
  typeName : Tc2_System.T_MaxString;
END_VAR
InitializeLogData();

symbolName := varInfo.Symbol;
typeName := varInfo.TypeName; 

format(
  sFormat := '%s [%s] : ',
  arg1 := Tc2_Utilities.F_STRING(symbolName),
  arg2 := Tc2_Utilities.F_STRING(typeName));
  
AppendString(format.sOut);
AppendAny(value);

AppendVariable REF= THIS^;
END_METHOD

/// Logs the log string in DEBUG level.
METHOD Debug : BOOL
VAR_INPUT
  /// Message to be appended to log string.
  message : Tc2_System.T_MaxString; 
END_VAR
InitializeLogData();
IF _logConditionSatisfied THEN
  IF _usedLogger <> InvalidLoggerReference THEN 
    _usedLogger.LogStandardFormat(Tc2_Standard.CONCAT(_logData, message), ShortenInstancePath(_instancePath), LogLevel.Debug); 
  ELSE
    Tc2_System.ADSLOGSTR(ADSLOG_MSGTYPE_LOG OR LogLevelToAdsLogMsgType(LogLevels.Error), 'usedLogger: No valid reference', ''); 
  END_IF
END_IF
_logDataInitialized := FALSE;
END_METHOD

/// Logs the log string in ERROR level.
METHOD Error : BOOL
VAR_INPUT
  /// Message to be appended to log string.
  message : Tc2_System.T_MaxString; 
END_VAR
InitializeLogData();
IF _logConditionSatisfied THEN
  IF _usedLogger <> InvalidLoggerReference THEN 
    _usedLogger.LogStandardFormat(Tc2_Standard.CONCAT(_logData, message), ShortenInstancePath(_instancePath), LogLevel.Error); 
  ELSE
    Tc2_System.ADSLOGSTR(ADSLOG_MSGTYPE_LOG OR LogLevelToAdsLogMsgType(LogLevels.Error), 'usedLogger: No valid reference', ''); 
  END_IF
END_IF
_logDataInitialized := FALSE;
END_METHOD

/// Logs the log string in FATAL level.
METHOD Fatal : BOOL
VAR_INPUT
  /// Message to be appended to log string.
  message : Tc2_System.T_MaxString; 
END_VAR
InitializeLogData();
IF _logConditionSatisfied THEN
  IF _usedLogger <> InvalidLoggerReference THEN 
    _usedLogger.LogStandardFormat(Tc2_Standard.CONCAT(_logData, message), ShortenInstancePath(_instancePath), LogLevel.Fatal); 
  ELSE
    Tc2_System.ADSLOGSTR(ADSLOG_MSGTYPE_LOG OR LogLevelToAdsLogMsgType(LogLevels.Error), 'usedLogger: No valid reference', ''); 
  END_IF
END_IF
_logDataInitialized := FALSE;
END_METHOD

/// Logs the log string in INFORMATION level.
METHOD Information : BOOL
VAR_INPUT
  /// Message to be appended to log string.
  message : Tc2_System.T_MaxString; 
END_VAR
InitializeLogData();
IF _logConditionSatisfied THEN
  IF _usedLogger <> InvalidLoggerReference THEN 
    _usedLogger.LogStandardFormat(Tc2_Standard.CONCAT(_logData, message), ShortenInstancePath(_instancePath), LogLevel.Information); 
  ELSE
    Tc2_System.ADSLOGSTR(ADSLOG_MSGTYPE_LOG OR LogLevelToAdsLogMsgType(LogLevels.Error), 'usedLogger: No valid reference', ''); 
  END_IF
END_IF
_logDataInitialized := FALSE;
END_METHOD

/// Initializes the reference to the core logger. Should only be called once from the core logger directly.
METHOD PUBLIC Init : BOOL
VAR_INPUT
  /// Reference to TcLoggerCore instance.
  ref2Core : ILogCore; 
END_VAR
IF s_loggerSingletonInstance = 0 THEN
	s_loggerSingletonInstance := ref2Core;
END_IF
END_METHOD

// Necessary to provide a fluent interface of the function. 
// Has to be called at the begin of any method that returns a reference to THIS^
METHOD PRIVATE InitializeLogData : BOOL
IF NOT _logDataInitialized THEN
  _logConditionSatisfied := TRUE;
  _logData := '';
  _logDataInitialized := TRUE;
  IF _usedLogger = 0 THEN _usedLogger := s_loggerSingletonInstance; END_IF
END_IF
END_METHOD

/// Conditional execution of the log command. Only executes logging when Cond = TRUE.
METHOD OnCondition : REFERENCE TO TcLog
VAR_INPUT
  /// Logs data only if this condition evaluates to TRUE.
  cond : BOOL; 
END_VAR
InitializeLogData();

_logConditionSatisfied := cond;

OnCondition REF= THIS^;
END_METHOD

/// Initializes the reference to the core logger. This enables you to use several
/// loggers with different configurations in one project.
METHOD SetLogger : BOOL
VAR_INPUT
  /// Reference to Core Logger
  ref2Core : ILogCore; 
END_VAR
_usedLogger := ref2Core;
END_METHOD

// Helper method. Shortens the instance path by omitting superfluent information
// such as concrete logger instance and plc/project names.
{attribute 'hide'}
METHOD PRIVATE ShortenInstancePath : Tc2_System.T_MaxString
VAR_INPUT
  path : Tc2_System.T_MaxString; // Instance path to be shortened.
END_VAR
VAR
  i : UINT;
  shortenedPath : Tc2_System.T_MaxString;
  positionInString : INT := 0;
  positionOfLastDot : INT := 0;
END_VAR
shortenedPath := path;

// Find last '.'
WHILE(Tc2_Standard.FIND(shortenedPath, '.') > 0) DO
  positionInString := Tc2_Standard.FIND(shortenedPath, '.');
  shortenedPath := Tc2_Standard.DELETE(shortenedPath, positionInString+1, 0); 
  positionOfLastDot := positionOfLastDot+positionInString;
END_WHILE

shortenedPath := Path;
// Delete instantiation of this FB (obvious information)
shortenedPath := Tc2_Standard.DELETE(shortenedPath, Tc2_Standard.LEN(shortenedPath)-positionOfLastDot+1, positionOfLastDot);
// Delete project information
positionInString := Tc2_Standard.FIND(shortenedPath, '.');
shortenedPath := Tc2_Standard.DELETE(shortenedPath, positionInString+1, 0);
// Delete PLC information
positionInString := Tc2_Standard.FIND(shortenedPath, '.');
shortenedPath := Tc2_Standard.DELETE(shortenedPath, positionInString+1, 0);

ShortenInstancePath := shortenedPath;
END_METHOD

/// Logs directly to ADS log, ignoring the settings of the base logger.
METHOD ToAdsLog : BOOL
VAR_INPUT
  /// Log level in which message should be logged to ADS.
  logLevel : LogLevels; 
END_VAR
InitializeLogData();

IF _logConditionSatisfied THEN
  Tc2_System.ADSLOGSTR(ADSLOG_MSGTYPE_LOG OR LogLevelToAdsLogMsgType(logLevel), _logData, ''); 
END_IF

_logDataInitialized := FALSE;
END_METHOD

/// Saves custom formatted log string. 
/// No addtitional information will be added, no formatting will be applied.
METHOD ToCustomFormat : BOOL
VAR_INPUT
  /// Message to be appended to log string.
  message : Tc2_System.T_MaxString; 
END_VAR
InitializeLogData();
IF _logConditionSatisfied THEN
  IF _usedLogger <> InvalidLoggerReference THEN 
    _usedLogger.LogCustomFormat(Tc2_Standard.CONCAT(_logData, message)); 
  ELSE
    Tc2_System.ADSLOGSTR(ADSLOG_MSGTYPE_LOG OR LogLevelToAdsLogMsgType(LogLevels.Error), 'usedLogger: No valid reference', ''); 
  END_IF
END_IF
_logDataInitialized := FALSE;
END_METHOD

/// Logs the log string in WARNING level.
METHOD Warning : BOOL
VAR_INPUT
  /// Message to be appended to log string.
  message : Tc2_System.T_MaxString; 
END_VAR
InitializeLogData();
IF _logConditionSatisfied THEN
  IF _usedLogger <> InvalidLoggerReference THEN 
    _usedLogger.LogStandardFormat(Tc2_Standard.CONCAT(_logData, message), ShortenInstancePath(_instancePath), LogLevel.Warning); 
  ELSE
    Tc2_System.ADSLOGSTR(ADSLOG_MSGTYPE_LOG OR LogLevelToAdsLogMsgType(LogLevels.Error), 'usedLogger: No valid reference', ''); 
  END_IF
END_IF
_logDataInitialized := FALSE;
END_METHOD

END_FUNCTION_BLOCK

// ---- Lib/TcLogCore.TcPOU
/// `TcLogCore` provides the base functionality of the logger and sets the configuration.
/// The logger can be configured by calling its methods that set the configuration.
///
/// > [!NOTE]
/// > `TcLogCore.RunLogger()` should be called once each cycle. The configuration methods should be called **before** 
/// > `RunLogger` is called.
///
/// When declaring an instance of TcLogCore, the ininital buffer size has to be set. If the buffer size is set too low, it will expand
/// automatically if enough memory is available.
///
/// To set the inital buffer size to accomodate 100 messages, use it like this:
///
/// ```st
/// VAR
///   myLogger: TcLogCore(BufferSize := 100 * (Tc2_System.MAX_STRING_LENGTH * Constants.FifoOverhead));
/// END_VAR
/// ```
///
{attribute 'hide_all_locals'}
FUNCTION_BLOCK TcLogCore IMPLEMENTS ILogCore
VAR
	_loggingSingleton : TcLog; // Logger-Singleton: Required to provide Singleton-functionality for TcLog.
	_utcTimeAsFileTime : Tc2_Utilities.T_FILETIME; // Current utc time as filetime
	_localTimeAsSystemTime : Tc2_Utilities.TIMESTRUCT; // Current local time as timestring
	_localTimeAsString : STRING; // Current local time as string
	_logCache : DynamicStringBuffer; // Dynamic string buffer to cache logs to be processed
	_startLoggingConfiguration : BOOL; // Aux variable to provide fluent interface.
	_internalErrorOccured : BOOL; // Aux variable to log internal errors to Error-property.                                                   				
	_config : LoggingConfiguration; // Logging configuration. Is set by invoking configuration methods.
	_error : Error; // Contains information about internal error.
	_busy : BOOL; // Logger is busy, typically with writing logs to the file system.
  _timeInfoReady : BOOL := FALSE; // Set to true once the time information is available
END_VAR

// Nothing to be done here. Logger works by invoking its methods.
// "RunLogger" contains all the implementation that has to be processed cyclically.

// Builds logging configuration.
// Required to provide a fluent interface.
// Has to be called at the begin of each method that configures the logger.
{attribute 'hide'}
METHOD PRIVATE BuildLoggingConfiguration : BOOL
IF NOT _startLoggingConfiguration THEN
	_startLoggingConfiguration := TRUE;
	
	_config.RollingInterval := RollingIntervals.Daily;
	_config.WriteToAds := FALSE;
	_config.FileName := '';
	_config.FilePath := 'c:\';
	_config.MinimumLevel := LogLevels.Debug;
	_config.Delimiter := '|';
	_config.IncludeInstancePath := FALSE;
	_config.LogFileLifespan := 0;
	_config.TimestampFormat := 'YYYYMMDD_hhmm_';
	_config.ValidTimestampsOnly := FALSE;
END_IF
END_METHOD

/// `Busy` evaluates to `TRUE` as long as the log file is kept open to append new log messages
/// or there are pending messages in the queue to be written to the logfile.
{attribute 'monitoring':='call'}
PROPERTY Busy : BOOL
GET
Busy := _busy;
END_GET
SET // PRIVATE
_busy := Busy;
END_SET
END_PROPERTY

/// Returns the current configuration of the logger.
{attribute 'monitoring':='variable'}
PROPERTY Configuration : LoggingConfiguration
GET
Configuration := _config;
END_GET
END_PROPERTY

/// Configuration method which sets the lifespan of log files. Once exceeded, they will be deleted.
METHOD DeleteLogFilesAfterDays : REFERENCE TO TcLogCore
VAR_INPUT
  /// Lifespan of logfiles in days.
	lifespan : UINT; 
END_VAR
BuildLoggingConfiguration();

_config.LogFileLifespan := lifespan;

DeleteLogFilesAfterDays REF= THIS^;
END_METHOD

/// Returns information about internal errors.
{attribute 'monitoring':='call'}
{attribute 'suppress_wrn_C0410'}
PROPERTY Error : REFERENCE TO Error
GET
Error REF= _error;
END_GET
END_PROPERTY

METHOD FB_init : BOOL
VAR_INPUT
	bInitRetains : BOOL; // if TRUE, the retain variables are initialized (warm start / cold start)
	bInCopyCode : BOOL; // if TRUE, the instance afterwards gets moved into the copy code (online change)
  /// Initial buffer size for the internal log message buffer
	bufferSize : UDINT;
END_VAR
_loggingSingleton.Init(THIS^);
_logCache.Init(bufferSize);
END_METHOD

/// Flushes the logging cache. All messages that have not yet been processed will be lost.
METHOD FlushCache : BOOL
_logCache.FlushCache();
END_METHOD

/// Configuration method. If this method is called, the instance path where the log 
/// messages has been triggered will be included in the log message. 
METHOD IncludeInstancePath : REFERENCE TO TcLogCore
BuildLoggingConfiguration();

_config.IncludeInstancePath := TRUE;

IncludeInstancePath REF= This^;
END_METHOD

/// Logger method. It should only be called from within objects that implement `ILog`.
/// Logs data in custom format. No additional formatting will be done. 
METHOD LogCustomFormat : BOOL
VAR_INPUT
  /// Data to be logged.
	data : Tc2_System.T_MaxString; 
END_VAR
IF(TimeInfoReady OR NOT _config.ValidTimestampsOnly) THEN 
	IF _config.WriteToAds THEN 
		Tc2_System.ADSLOGSTR(ADSLOG_MSGTYPE_LOG OR ADSLOG_MSGTYPE_HINT, data, ''); 
	END_IF
	
	IF _config.file_name <> '' THEN 
		_logCache.AddLine(data);
	END_IF
END_IF
END_METHOD

/// Logger method. It should only be called from within objects that implement `ILog`.
/// Logs in the standard format. This includes
/// - timestamp
/// - log level
/// - log message
/// - instance path of logging source (optional)
/// The message will only be logged if the logging level exceeds the configured minimum logging level.
METHOD LogStandardFormat : BOOL
VAR_INPUT
  /// Data to be logged.
	data : Tc2_System.T_MaxString; 
  /// Instance path of calling logger to locate source of logging message.
	instancePath : Tc2_System.T_MaxString;
  /// Log level of message. 
	logLevel : LogLevels; 
END_VAR
VAR_INST
  {attribute 'hide'}
	messageBuilder : StringBuilder;
END_VAR
IF LogLevel >= _config.MinimumLevel AND (TimeInfoReady OR NOT _config.ValidTimestampsOnly)  THEN
	IF _config.WriteToAds THEN 
		Tc2_System.ADSLOGSTR(
			ADSLOG_MSGTYPE_LOG OR LogLevelToAdsLogMsgType(logLevel), 
			messageBuilder
				.Reset()
				.AppendIf(_config.IncludeInstancePath, instancePath)
				.AppendIf(_config.IncludeInstancePath, _config.Delimiter)
				.Append(data)
				.ToString(), 
			''
		); 
	END_IF
	
	IF _config.file_name <> '' THEN 
		_logCache.AddLine(
			messageBuilder
					.Reset()
					.Append(_localTimeAsString)
					.Append(_config.Delimiter)
					.Append(TO_STRING(LogLevel))
					.AppendIf(_config.IncludeInstancePath, _config.Delimiter)
					.AppendIf(_config.IncludeInstancePath, instancePath)
					.Append(_config.Delimiter)
					.Append(data)
					.ToString()
		);
	END_IF
END_IF
END_METHOD

/// Configuration method.
/// Sets the minimum log level. Log messages below this level 
/// will not be logged.
METHOD MinimumLevel : REFERENCE TO TcLogCore
VAR_INPUT
  /// Minimum log level to be logged.
	level : LogLevel; 
END_VAR
BuildLoggingConfiguration();

_config.MinimumLevel := level;

MinimumLevel REF=THIS^;
END_METHOD

// Checks the specified rolling interval for the file name.
// Generates new file name if rolling intervall exceeded.
{attribute 'hide_all_locals'}
{attribute 'hide'}
METHOD PRIVATE RollingIntervalReached : BOOL
VAR_INPUT
	currentUtcTime : Tc2_Utilities.TIMESTRUCT;  // Current system time as utc
	rollingInterval : RollingIntervals; // Rolling interval 
END_VAR
VAR_INST
	newHour : Tc2_Standard.R_TRIG;
	newDay : Tc2_Standard.R_TRIG;
	newMonth : Tc2_Standard.R_TRIG;
	
	hourRolled : BOOL;
	dayRolled : BOOL;
	monthRolled : BOOL;
END_VAR
newHour(CLK := (currentUtcTime.wMinute = 0 AND currentUtcTime.wSecond = 0), 
	Q => hourRolled);
newDay(CLK := (hourRolled AND currentUtcTime.wHour = 0), 
	Q => dayRolled);
newMonth(CLK := (dayRolled AND currentUtcTime.wDay = 1), 
	Q => monthRolled);

RollingIntervalReached := 	(hourRolled 	AND rollingInterval = RollingIntervals.Hourly) OR
							(dayRolled 		AND rollingInterval = RollingIntervals.Daily) 	OR
							(monthRolled 	AND rollingInterval = RollingIntervals.Monthly);
END_METHOD

/// Cyclic method of Logger.
/// This method has to be executed in every plc cycle and runs 
/// all internal methods that have to be executed cyclically.
/// > [!NOTE]
/// > This method should be the last method of `TcLogCore` to be called in each cycle.
{attribute 'hide_all_locals'}
METHOD RunLogger : BOOL
VAR_INST
	newDay : Tc2_Standard.R_TRIG; 
	dateTime : DateTime;
	deleteExpiredLogFiles : DeleteOldFiles;
	fileNameStringBuilder : StringBuilder;
	timeStamp : STRING; // Timestamp used for filename
END_VAR
// Generate time data (shared state)
dateTime();
IF dateTime.Done THEN _timeInfoReady := TRUE; END_IF

_localTimeAsSystemTime := dateTime.AsLocalSystemTime;
_localTimeAsString := dateTime.AsLocalSystemTimeString;
_utcTimeAsFileTime := dateTime.AsUtcFileTime;

// Generate new timestamp for filename
IF RollingIntervalReached(_localTimeAsSystemTime, _config.RollingInterval) OR dateTime.Done THEN
	timeStamp := dateTime.ToFormatString(_config.TimestampFormat);
END_IF

// Delete expired log files
newDay(CLK := _localTimeAsSystemTime.wHour = 0);
deleteExpiredLogFiles(
	StartScan 			:= 	newDay.Q AND (_config.LogFileLifespan > 0),
	ExpirationInDays 	:=	_config.LogFileLifespan,
	FilePath			:=	_config.file_path,
	FileName 			:=	_config.file_name,
	CurrentUtcTime 		:= 	_utcTimeAsFileTime	
	);
IF deleteExpiredLogFiles.Error.Active THEN
	_internalErrorOccured := TRUE;
	_error := deleteExpiredLogFiles.Error;
END_IF
		
// Persist logging messages to file
_logCache.PersistToFile(
  TimeInfoReady,
	fileNameStringBuilder
		.Reset()
		.Append(_config.file_path)
		.AppendIf(Tc2_Standard.RIGHT(_config.FilePath, 1) <> '\', '\')
		.Append(timeStamp)
		.Append(_config.file_name)
		.ToString()
);
IF _logCache.Error.Active THEN
	_internalErrorOccured := TRUE;
	_error := _logCache.Error;
END_IF

// Forward busy state of LogCache 
Busy := _logCache.Busy;

// Reset Logging configuration: neccesary in order to provide fluent interface
_startLoggingConfiguration := FALSE;

// Reset error flag each cycle to automatically confirm errors once they are gone.
IF NOT _internalErrorOccured THEN
	_error.Active := FALSE;
	_error.Code := ErrorCodes.None;
	_error.Info := '';
END_IF
_internalErrorOccured := FALSE;
END_METHOD

/// Configuration method
/// Sets delimiter between different columns of log file.
METHOD SetDelimiter : REFERENCE TO TcLogCore
VAR_INPUT
  /// Delimiter between different columns of log file.
	delimiter : STRING(1); 
END_VAR
BuildLoggingConfiguration();

_config.Delimiter := delimiter;

SetDelimiter REF=THIS^;
END_METHOD

/// Configuration method.
/// Sets the rolling interval of the log file. Once the rolling interval
/// expires, a file name with a new timestamp will be generated.
METHOD SetRollingInterval : REFERENCE TO TcLogCore
VAR_INPUT
  /// Rolling interval for log file. Once exceeded, a new log file will be created.
	interval : RollingIntervals; 
END_VAR
BuildLoggingConfiguration();

_config.RollingInterval := interval;

SetRollingInterval REF= THIS^;
END_METHOD

/// `TimeInfoReady` evaluates to `TRUE` once the time information used by determine
/// the timestamp for the message is available.
{attribute 'monitoring':='call'}
PROPERTY TimeInfoReady : BOOL
GET
TimeInfoReady := _timeInfoReady;
END_GET
END_PROPERTY

/// Configuration method.
/// Sets the format of the timestamp in the file name. 
/// 
/// The following format options are available:
///	Y : year
///	M : month
/// D : day
/// h : hour 
/// m : minute
/// s : second
/// i : millisecond
/// 
/// Example: _YYMMDD-hh:mm:ss:iii_
/// => _20210812-12:30:22:123_
METHOD TimestampFormat : REFERENCE TO TcLogCore
VAR_INPUT
  /// Format the timestamp should have.
	format : STRING; 
END_VAR
BuildLoggingConfiguration();

_config.TimestampFormat := format;

TimestampFormat REF= THIS^;
END_METHOD

/// Configuration method. If this method is called, only valid timestamps are logged.
/// Note that using this configuration will skip logging anything during the first few PLC cycles, 
/// as TwinCAT needs a few cycles to initialize its time information.
METHOD ValidTimestampsOnly : REFERENCE TO TcLogCore
BuildLoggingConfiguration();

_config.ValidTimestampsOnly := TRUE;

ValidTimestampsOnly REF= This^;
END_METHOD

/// Configuration method.
/// If this method is called, the logs will be written to ADS.
METHOD WriteToAds : REFERENCE TO TcLogCore
BuildLoggingConfiguration();

_config.WriteToAds := TRUE;

WriteToAds REF= This^;
END_METHOD

/// Configuration method.
/// If this method is called, the logs will be persisted to the file system.
METHOD WriteToFile : REFERENCE TO TcLogCore
VAR_INPUT
  /// File path the logs will be written to.
	path : Tc2_System.T_MaxString; 
  /// File name of the log file. Will automatically be prefixed by timestamp.
	fileName : STRING; 
END_VAR
BuildLoggingConfiguration();

IF Tc2_Standard.RIGHT(path, 1) <> '\' THEN
  _config.file_path := TC2_Standard.CONCAT(path, '\');  
ELSE
  _config.file_path := path;
END_IF
_config.file_name := fileName;

WriteToFile REF= This^;
END_METHOD

END_FUNCTION_BLOCK

// ---- Lib/TcLogTrig.TcPOU
/// This function block can be used to log on rising or falling edges.
/// For each signal that should be watched, a separate instance of `TcLogTrig` 
/// must be created.
FUNCTION_BLOCK TcLogTrig EXTENDS TcLog

/// Logs data on falling edge of `CLK`.
{attribute 'hide_all_locals'}
METHOD OnFallingEdge : REFERENCE TO TcLog
VAR_INPUT
  /// Falling edge triggers logging the data.
  CLK : BOOL; 
END_VAR
VAR_INST
    fTrig : Tc2_Standard.F_TRIG;
END_VAR
fTrig(CLK:=CLK);

SUPER^.OnCondition(fTrig.Q);

OnFallingEdge REF= THIS^;
END_METHOD

/// Logs data on rising edge of `CLK`.
{attribute 'hide_all_locals'}
METHOD OnRisingEdge : REFERENCE TO TcLog
VAR_INPUT
  /// Rising edge logs data.
  CLK : BOOL; 
END_VAR
VAR_INST
    rTrig : Tc2_Standard.R_TRIG;
END_VAR
rTrig(CLK:=CLK);

SUPER^.OnCondition(rTrig.Q);

OnRisingEdge REF= THIS^;
END_METHOD

END_FUNCTION_BLOCK
